// TIA Portal V19 export
DATA_BLOCK "Decoiler2_PERS"   // DB54
// stored: MemoryReserve 100
   VAR RETAIN
      PersistentValues : "Decoiler_Pers";
   END_VAR
BEGIN
   PersistentValues.CoilDiamSensor.Data.AnalogicSensor_OffsetValue := -3794.985;
   PersistentValues.CoilDiamSensor.Data.AnalogicSensor_OffsetValid := TRUE;
   PersistentValues.CoilDiamSensor.Par.AnalogicSensor_Enable := TRUE;
   PersistentValues.CoilDiamSensor.Par.AnalogicSensor_RangeLow := 3000.0;
   PersistentValues.CoilDiamSensor.Par.AnalogicSensor_RangeHigh := 0.0;
   PersistentValues.CoilDiamSensor.Par.Diam_Min := 500.0;
   PersistentValues.CoilDiamSensor.Par.Diam_Max := 1800.0;
   PersistentValues.CoilDiamSensor.Par.EndCoil_Diam := 510.0;
   PersistentValues.CoilDiamSensor.Par.EndCoil_Timer := T#3S;
   PersistentValues.Loop.Par.DelayRestartAfterMaxLoop := T#500MS;
   PersistentValues.Loop.Par.DelayStopMaxLoop := T#500MS;
   PersistentValues.Loop.Par.SensoAdjVel_PercentageMinus := 2.0;
   PersistentValues.Loop.Par.SensoAdjVel_PercentagePlus := 10.0;
   PersistentValues.Loop.Par.SensoAdjVel_PercentagePlusPlus := 30.0;
   PersistentValues.Loop.Par.SensoAdjVel_DelayPlusPlus := T#10S;
   PersistentValues.Feed.Man.VelBwd := 3000.0;
   PersistentValues.Feed.Man.VelFwdHigh := 3000.0;
   PersistentValues.Feed.Man.VelFwdLow := 3000.0;
   PersistentValues.Feed.Man.Acc := 500.0;
   PersistentValues.Feed.Man.Dec := 500.0;
   PersistentValues.Feed.Man.DelayChangeVel := T#1MS;
   PersistentValues.Coupling.Engaged := TRUE;
   PersistentValues.Jaws.Par.Pause := T#10M;
   PersistentValues.Jaws.Par.Duration := T#5S;
   PersistentValues.Jaws.Par.DiamEnable := 550.0;
   PersistentValues.PneumaticBracking.DiameterChangeBrake := 600.0;
END_DATA_BLOCK
